Staubli VAL3: fbkStreamer.pgx

public program fbkStreamer()
begin

end
